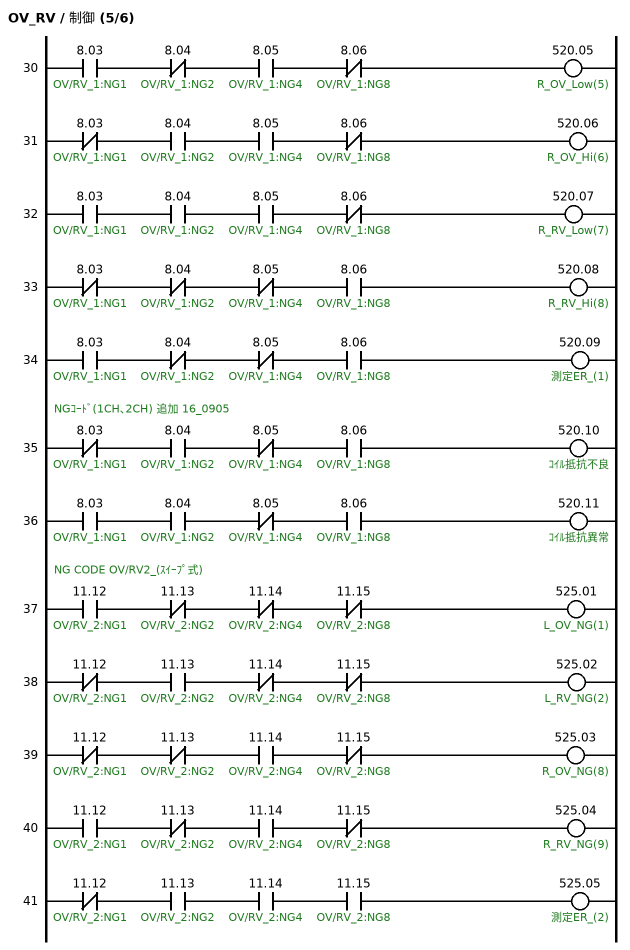
; [picture p120: OV_RV / 制御, rungs 30-41]
; rung 30
LD 8.03  ; OV/RV_1:NG1
ANDNOT 8.04  ; OV/RV_1:NG2
AND 8.05  ; OV/RV_1:NG4
ANDNOT 8.06  ; OV/RV_1:NG8
OUT 520.05  ; R_OV_Low(5)
; rung 31
LDNOT 8.03  ; OV/RV_1:NG1
AND 8.04  ; OV/RV_1:NG2
AND 8.05  ; OV/RV_1:NG4
ANDNOT 8.06  ; OV/RV_1:NG8
OUT 520.06  ; R_OV_Hi(6)
; rung 32
LD 8.03  ; OV/RV_1:NG1
AND 8.04  ; OV/RV_1:NG2
AND 8.05  ; OV/RV_1:NG4
ANDNOT 8.06  ; OV/RV_1:NG8
OUT 520.07  ; R_RV_Low(7)
; rung 33
LDNOT 8.03  ; OV/RV_1:NG1
ANDNOT 8.04  ; OV/RV_1:NG2
ANDNOT 8.05  ; OV/RV_1:NG4
AND 8.06  ; OV/RV_1:NG8
OUT 520.08  ; R_RV_Hi(8)
; rung 34
LD 8.03  ; OV/RV_1:NG1
ANDNOT 8.04  ; OV/RV_1:NG2
ANDNOT 8.05  ; OV/RV_1:NG4
AND 8.06  ; OV/RV_1:NG8
OUT 520.09  ; 測定ER_(1)
; rung 35: NGｺｰﾄﾞ(1CH､2CH) 追加 16_0905
LDNOT 8.03  ; OV/RV_1:NG1
AND 8.04  ; OV/RV_1:NG2
ANDNOT 8.05  ; OV/RV_1:NG4
AND 8.06  ; OV/RV_1:NG8
OUT 520.10  ; ｺｲﾙ抵抗不良
; rung 36
LD 8.03  ; OV/RV_1:NG1
AND 8.04  ; OV/RV_1:NG2
ANDNOT 8.05  ; OV/RV_1:NG4
AND 8.06  ; OV/RV_1:NG8
OUT 520.11  ; ｺｲﾙ抵抗異常
; rung 37: NG CODE OV/RV2_(ｽｲｰﾌﾟ式)
LD 11.12  ; OV/RV_2:NG1
ANDNOT 11.13  ; OV/RV_2:NG2
ANDNOT 11.14  ; OV/RV_2:NG4
ANDNOT 11.15  ; OV/RV_2:NG8
OUT 525.01  ; L_OV_NG(1)
; rung 38
LDNOT 11.12  ; OV/RV_2:NG1
AND 11.13  ; OV/RV_2:NG2
ANDNOT 11.14  ; OV/RV_2:NG4
ANDNOT 11.15  ; OV/RV_2:NG8
OUT 525.02  ; L_RV_NG(2)
; rung 39
LDNOT 11.12  ; OV/RV_2:NG1
ANDNOT 11.13  ; OV/RV_2:NG2
AND 11.14  ; OV/RV_2:NG4
ANDNOT 11.15  ; OV/RV_2:NG8
OUT 525.03  ; R_OV_NG(8)
; rung 40
LD 11.12  ; OV/RV_2:NG1
ANDNOT 11.13  ; OV/RV_2:NG2
AND 11.14  ; OV/RV_2:NG4
ANDNOT 11.15  ; OV/RV_2:NG8
OUT 525.04  ; R_RV_NG(9)
; rung 41
LDNOT 11.12  ; OV/RV_2:NG1
AND 11.13  ; OV/RV_2:NG2
AND 11.14  ; OV/RV_2:NG4
AND 11.15  ; OV/RV_2:NG8
OUT 525.05  ; 測定ER_(2)

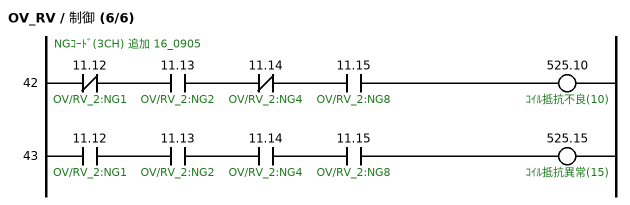
; rung 42: NGｺｰﾄﾞ(3CH) 追加 16_0905
LDNOT 11.12  ; OV/RV_2:NG1
AND 11.13  ; OV/RV_2:NG2
ANDNOT 11.14  ; OV/RV_2:NG4
AND 11.15  ; OV/RV_2:NG8
OUT 525.10  ; ｺｲﾙ抵抗不良(10)
; rung 43
LD 11.12  ; OV/RV_2:NG1
AND 11.13  ; OV/RV_2:NG2
AND 11.14  ; OV/RV_2:NG4
AND 11.15  ; OV/RV_2:NG8
OUT 525.15  ; ｺｲﾙ抵抗異常(15)

### Section 出力

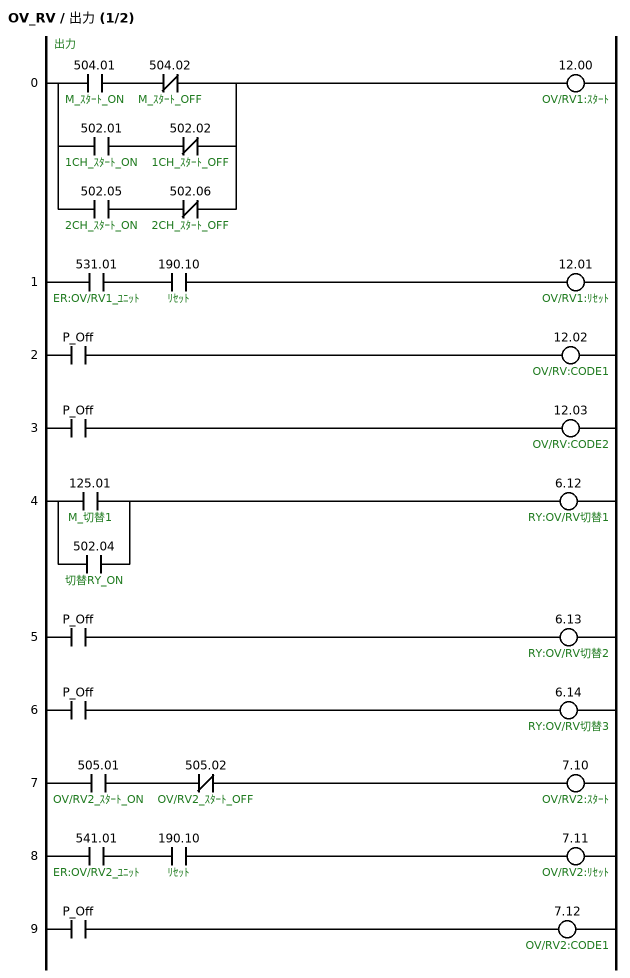
; rung 0: 出力
LD 504.01  ; M_ｽﾀｰﾄ_ON
ANDNOT 504.02  ; M_ｽﾀｰﾄ_OFF
LD 502.01  ; 1CH_ｽﾀｰﾄ_ON
ANDNOT 502.02  ; 1CH_ｽﾀｰﾄ_OFF
ORLD
LD 502.05  ; 2CH_ｽﾀｰﾄ_ON
ANDNOT 502.06  ; 2CH_ｽﾀｰﾄ_OFF
ORLD
OUT 12.00  ; OV/RV1:ｽﾀｰﾄ
; rung 1
LD 531.01  ; ER:OV/RV1_ﾕﾆｯﾄ
AND 190.10  ; ﾘｾｯﾄ
OUT 12.01  ; OV/RV1:ﾘｾｯﾄ
; rung 2
LD P_Off
OUT 12.02  ; OV/RV:CODE1
; rung 3
LD P_Off
OUT 12.03  ; OV/RV:CODE2
; rung 4
LD 125.01  ; M_切替1
OR 502.04  ; 切替RY_ON
OUT 6.12  ; RY:OV/RV切替1
; rung 5
LD P_Off
OUT 6.13  ; RY:OV/RV切替2
; rung 6
LD P_Off
OUT 6.14  ; RY:OV/RV切替3
; rung 7
LD 505.01  ; OV/RV2_ｽﾀｰﾄ_ON
ANDNOT 505.02  ; OV/RV2_ｽﾀｰﾄ_OFF
OUT 7.10  ; OV/RV2:ｽﾀｰﾄ
; rung 8
LD 541.01  ; ER:OV/RV2_ﾕﾆｯﾄ
AND 190.10  ; ﾘｾｯﾄ
OUT 7.11  ; OV/RV2:ﾘｾｯﾄ
; rung 9
LD P_Off
OUT 7.12  ; OV/RV2:CODE1

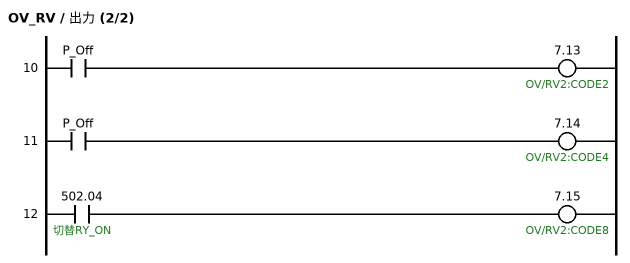
; rung 10
LD P_Off
OUT 7.13  ; OV/RV2:CODE2
; rung 11
LD P_Off
OUT 7.14  ; OV/RV2:CODE4
; rung 12
LD 502.04  ; 切替RY_ON
OUT 7.15  ; OV/RV2:CODE8

### Section ｴﾗｰ

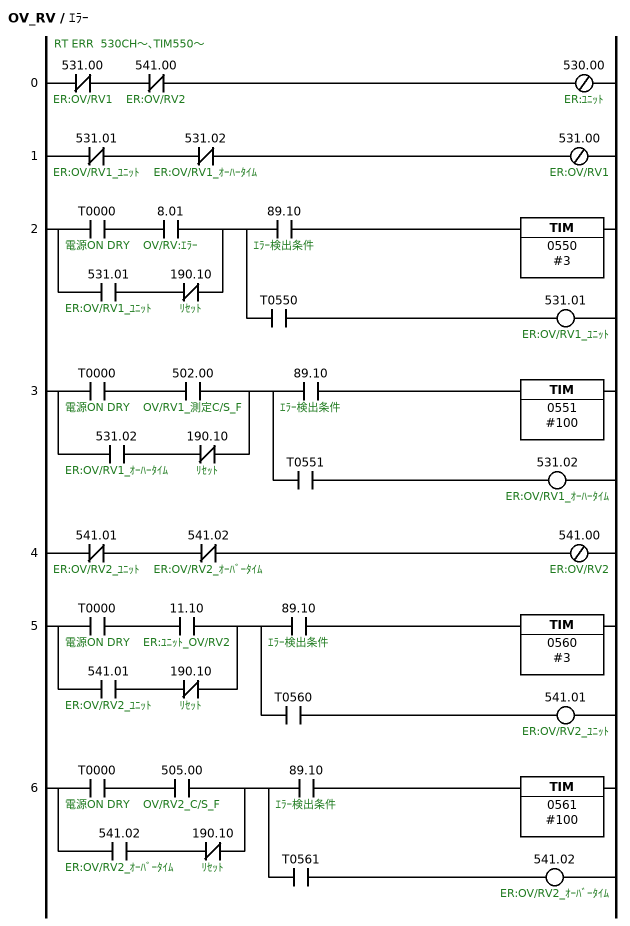
; rung 0: RT ERR  530CH～､TIM550～
LDNOT 531.00  ; ER:OV/RV1
ANDNOT 541.00  ; ER:OV/RV2
OUTNOT 530.00  ; ER:ﾕﾆｯﾄ
; rung 1
LDNOT 531.01  ; ER:OV/RV1_ﾕﾆｯﾄ
ANDNOT 531.02  ; ER:OV/RV1_ｵｰﾊｰﾀｲﾑ
OUTNOT 531.00  ; ER:OV/RV1
; rung 2
LD T0000  ; 電源ON DRY
AND 8.01  ; OV/RV:ｴﾗｰ
LD 531.01  ; ER:OV/RV1_ﾕﾆｯﾄ
ANDNOT 190.10  ; ﾘｾｯﾄ
ORLD
OUT TR0
AND 89.10  ; ｴﾗｰ検出条件
TIM 0550 #3
LD TR0
AND T0550
OUT 531.01  ; ER:OV/RV1_ﾕﾆｯﾄ
; rung 3
LD T0000  ; 電源ON DRY
AND 502.00  ; OV/RV1_測定C/S_F
LD 531.02  ; ER:OV/RV1_ｵｰﾊｰﾀｲﾑ
ANDNOT 190.10  ; ﾘｾｯﾄ
ORLD
OUT TR0
AND 89.10  ; ｴﾗｰ検出条件
TIM 0551 #100
LD TR0
AND T0551
OUT 531.02  ; ER:OV/RV1_ｵｰﾊｰﾀｲﾑ
; rung 4
LDNOT 541.01  ; ER:OV/RV2_ﾕﾆｯﾄ
ANDNOT 541.02  ; ER:OV/RV2_ｵｰﾊﾞｰﾀｲﾑ
OUTNOT 541.00  ; ER:OV/RV2
; rung 5
LD T0000  ; 電源ON DRY
AND 11.10  ; ER:ﾕﾆｯﾄ_OV/RV2
LD 541.01  ; ER:OV/RV2_ﾕﾆｯﾄ
ANDNOT 190.10  ; ﾘｾｯﾄ
ORLD
OUT TR0
AND 89.10  ; ｴﾗｰ検出条件
TIM 0560 #3
LD TR0
AND T0560
OUT 541.01  ; ER:OV/RV2_ﾕﾆｯﾄ
; rung 6
LD T0000  ; 電源ON DRY
AND 505.00  ; OV/RV2_C/S_F
LD 541.02  ; ER:OV/RV2_ｵｰﾊﾞｰﾀｲﾑ
ANDNOT 190.10  ; ﾘｾｯﾄ
ORLD
OUT TR0
AND 89.10  ; ｴﾗｰ検出条件
TIM 0561 #100
LD TR0
AND T0561
OUT 541.02  ; ER:OV/RV2_ｵｰﾊﾞｰﾀｲﾑ

### Section END
; rung 0
END(001)

## Program CP (cyclic task 5)

### Section 制御

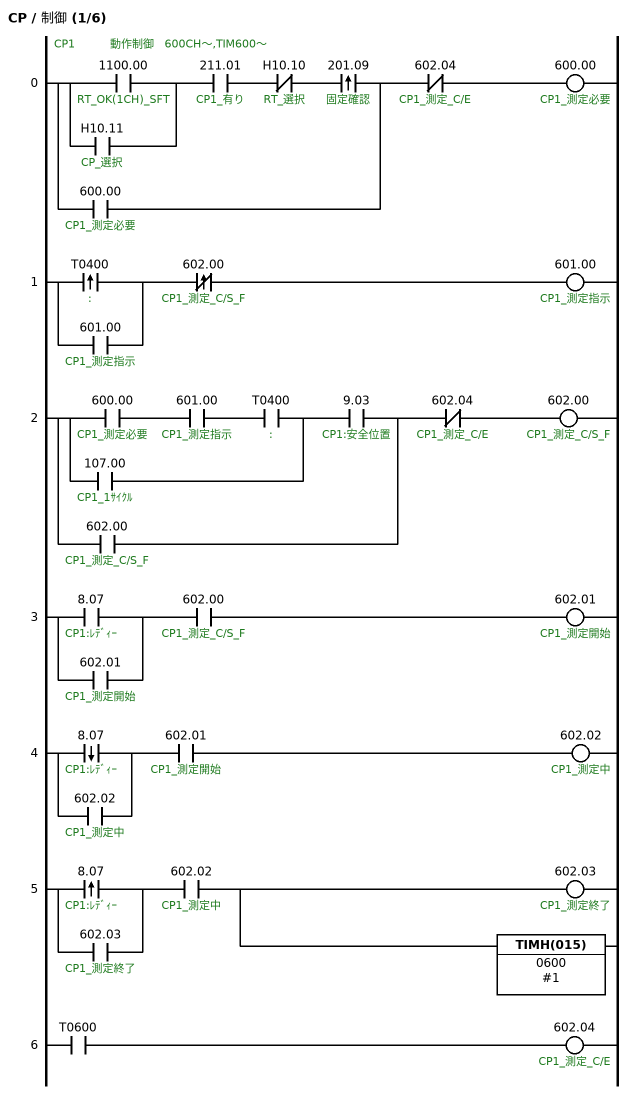
; rung 0: CP1          動作制御   600CH～,TIM600～
LD 1100.00  ; RT_OK(1CH)_SFT
OR H10.11  ; CP_選択
AND 211.01  ; CP1_有り
ANDNOT H10.10  ; RT_選択
@AND 201.09  ; 固定確認
OR 600.00  ; CP1_測定必要
ANDNOT 602.04  ; CP1_測定_C/E
OUT 600.00  ; CP1_測定必要
; rung 1
@LD T0400  ; :
OR 601.00  ; CP1_測定指示
@ANDNOT 602.00  ; CP1_測定_C/S_F
OUT 601.00  ; CP1_測定指示
; rung 2
LD 600.00  ; CP1_測定必要
AND 601.00  ; CP1_測定指示
AND T0400  ; :
OR 107.00  ; CP1_1ｻｲｸﾙ
AND 9.03  ; CP1:安全位置
OR 602.00  ; CP1_測定_C/S_F
ANDNOT 602.04  ; CP1_測定_C/E
OUT 602.00  ; CP1_測定_C/S_F
; rung 3
LD 8.07  ; CP1:ﾚﾃﾞｨｰ
OR 602.01  ; CP1_測定開始
AND 602.00  ; CP1_測定_C/S_F
OUT 602.01  ; CP1_測定開始
; rung 4
%LD 8.07  ; CP1:ﾚﾃﾞｨｰ
OR 602.02  ; CP1_測定中
AND 602.01  ; CP1_測定開始
OUT 602.02  ; CP1_測定中
; rung 5
@LD 8.07  ; CP1:ﾚﾃﾞｨｰ
OR 602.03  ; CP1_測定終了
AND 602.02  ; CP1_測定中
OUT 602.03  ; CP1_測定終了
TIMH(015) 0600 #1
; rung 6
LD T0600
OUT 602.04  ; CP1_測定_C/E

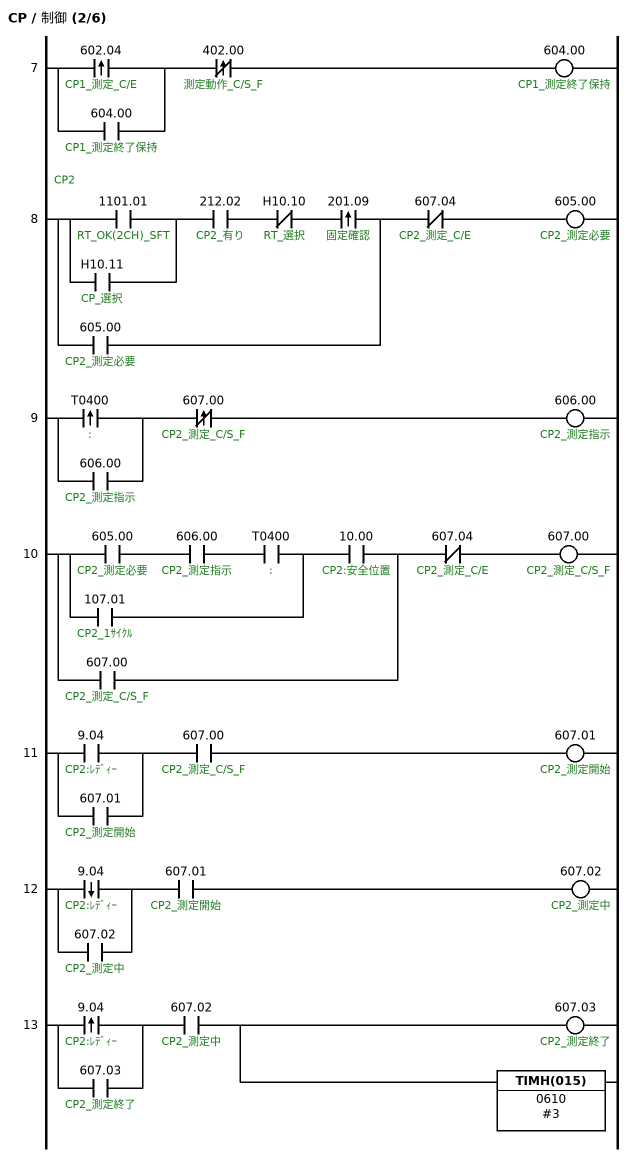
; rung 7
@LD 602.04  ; CP1_測定_C/E
OR 604.00  ; CP1_測定終了保持
@ANDNOT 402.00  ; 測定動作_C/S_F
OUT 604.00  ; CP1_測定終了保持
; rung 8: CP2
LD 1101.01  ; RT_OK(2CH)_SFT
OR H10.11  ; CP_選択
AND 212.02  ; CP2_有り
ANDNOT H10.10  ; RT_選択
@AND 201.09  ; 固定確認
OR 605.00  ; CP2_測定必要
ANDNOT 607.04  ; CP2_測定_C/E
OUT 605.00  ; CP2_測定必要
; rung 9
@LD T0400  ; :
OR 606.00  ; CP2_測定指示
@ANDNOT 607.00  ; CP2_測定_C/S_F
OUT 606.00  ; CP2_測定指示
; rung 10
LD 605.00  ; CP2_測定必要
AND 606.00  ; CP2_測定指示
AND T0400  ; :
OR 107.01  ; CP2_1ｻｲｸﾙ
AND 10.00  ; CP2:安全位置
OR 607.00  ; CP2_測定_C/S_F
ANDNOT 607.04  ; CP2_測定_C/E
OUT 607.00  ; CP2_測定_C/S_F
; rung 11
LD 9.04  ; CP2:ﾚﾃﾞｨｰ
OR 607.01  ; CP2_測定開始
AND 607.00  ; CP2_測定_C/S_F
OUT 607.01  ; CP2_測定開始
; rung 12
%LD 9.04  ; CP2:ﾚﾃﾞｨｰ
OR 607.02  ; CP2_測定中
AND 607.01  ; CP2_測定開始
OUT 607.02  ; CP2_測定中
; rung 13
@LD 9.04  ; CP2:ﾚﾃﾞｨｰ
OR 607.03  ; CP2_測定終了
AND 607.02  ; CP2_測定中
OUT 607.03  ; CP2_測定終了
TIMH(015) 0610 #3

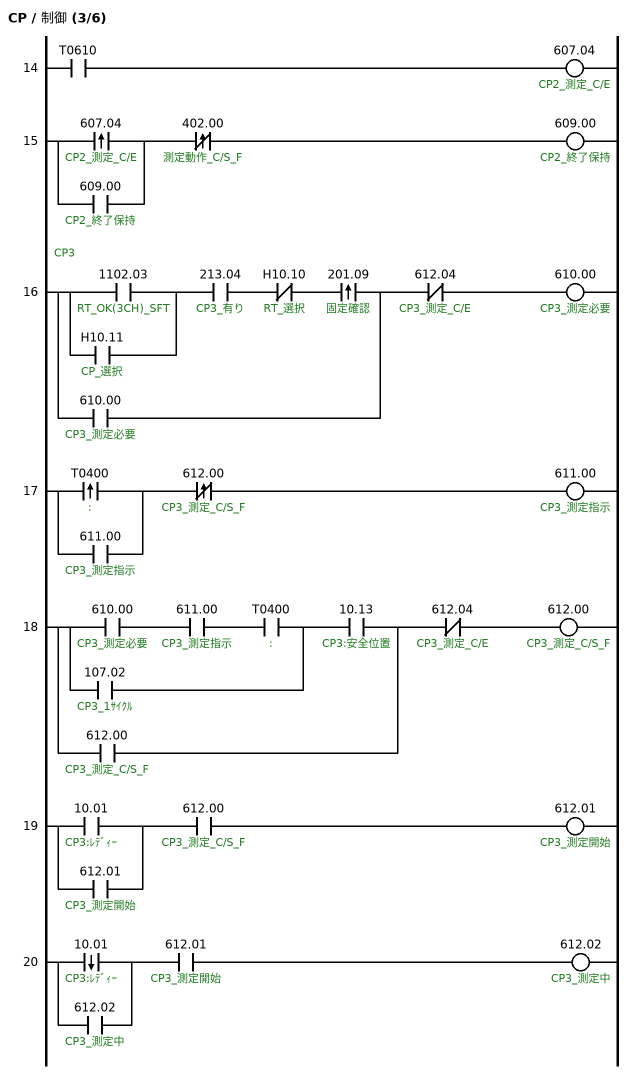
; rung 14
LD T0610
OUT 607.04  ; CP2_測定_C/E
; rung 15
@LD 607.04  ; CP2_測定_C/E
OR 609.00  ; CP2_終了保持
@ANDNOT 402.00  ; 測定動作_C/S_F
OUT 609.00  ; CP2_終了保持
; rung 16: CP3
LD 1102.03  ; RT_OK(3CH)_SFT
OR H10.11  ; CP_選択
AND 213.04  ; CP3_有り
ANDNOT H10.10  ; RT_選択
@AND 201.09  ; 固定確認
OR 610.00  ; CP3_測定必要
ANDNOT 612.04  ; CP3_測定_C/E
OUT 610.00  ; CP3_測定必要
; rung 17
@LD T0400  ; :
OR 611.00  ; CP3_測定指示
@ANDNOT 612.00  ; CP3_測定_C/S_F
OUT 611.00  ; CP3_測定指示
; rung 18
LD 610.00  ; CP3_測定必要
AND 611.00  ; CP3_測定指示
AND T0400  ; :
OR 107.02  ; CP3_1ｻｲｸﾙ
AND 10.13  ; CP3:安全位置
OR 612.00  ; CP3_測定_C/S_F
ANDNOT 612.04  ; CP3_測定_C/E
OUT 612.00  ; CP3_測定_C/S_F
; rung 19
LD 10.01  ; CP3:ﾚﾃﾞｨｰ
OR 612.01  ; CP3_測定開始
AND 612.00  ; CP3_測定_C/S_F
OUT 612.01  ; CP3_測定開始
; rung 20
%LD 10.01  ; CP3:ﾚﾃﾞｨｰ
OR 612.02  ; CP3_測定中
AND 612.01  ; CP3_測定開始
OUT 612.02  ; CP3_測定中

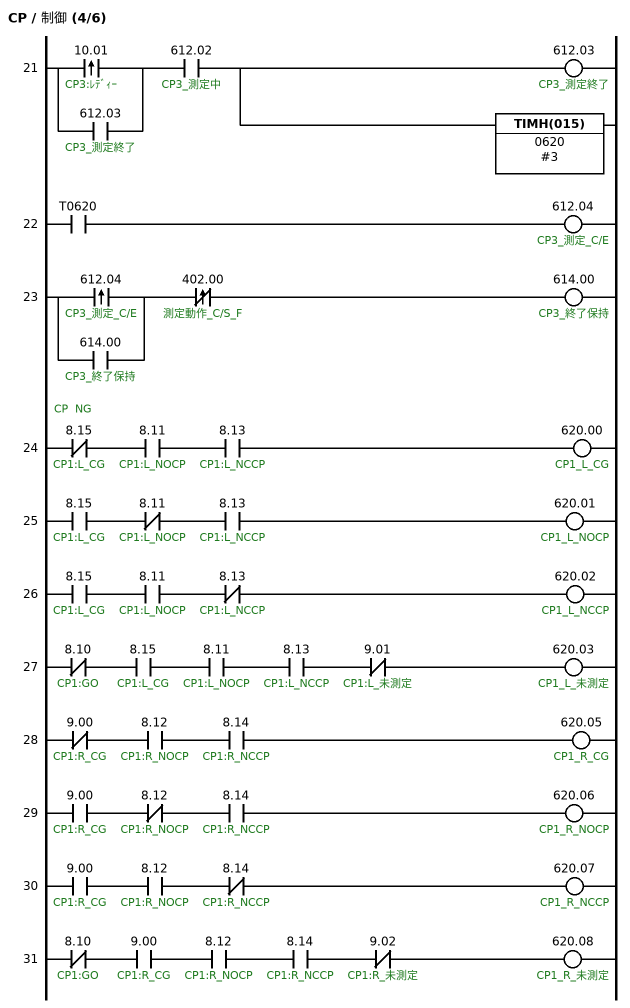
; rung 21
@LD 10.01  ; CP3:ﾚﾃﾞｨｰ
OR 612.03  ; CP3_測定終了
AND 612.02  ; CP3_測定中
OUT 612.03  ; CP3_測定終了
TIMH(015) 0620 #3
; rung 22
LD T0620
OUT 612.04  ; CP3_測定_C/E
; rung 23
@LD 612.04  ; CP3_測定_C/E
OR 614.00  ; CP3_終了保持
@ANDNOT 402.00  ; 測定動作_C/S_F
OUT 614.00  ; CP3_終了保持
; rung 24: CP  NG
LDNOT 8.15  ; CP1:L_CG
AND 8.11  ; CP1:L_NOCP
AND 8.13  ; CP1:L_NCCP
OUT 620.00  ; CP1_L_CG
; rung 25
LD 8.15  ; CP1:L_CG
ANDNOT 8.11  ; CP1:L_NOCP
AND 8.13  ; CP1:L_NCCP
OUT 620.01  ; CP1_L_NOCP
; rung 26
LD 8.15  ; CP1:L_CG
AND 8.11  ; CP1:L_NOCP
ANDNOT 8.13  ; CP1:L_NCCP
OUT 620.02  ; CP1_L_NCCP
; rung 27
LDNOT 8.10  ; CP1:GO
AND 8.15  ; CP1:L_CG
AND 8.11  ; CP1:L_NOCP
AND 8.13  ; CP1:L_NCCP
ANDNOT 9.01  ; CP1:L_未測定
OUT 620.03  ; CP1_L_未測定
; rung 28
LDNOT 9.00  ; CP1:R_CG
AND 8.12  ; CP1:R_NOCP
AND 8.14  ; CP1:R_NCCP
OUT 620.05  ; CP1_R_CG
; rung 29
LD 9.00  ; CP1:R_CG
ANDNOT 8.12  ; CP1:R_NOCP
AND 8.14  ; CP1:R_NCCP
OUT 620.06  ; CP1_R_NOCP
; rung 30
LD 9.00  ; CP1:R_CG
AND 8.12  ; CP1:R_NOCP
ANDNOT 8.14  ; CP1:R_NCCP
OUT 620.07  ; CP1_R_NCCP
; rung 31
LDNOT 8.10  ; CP1:GO
AND 9.00  ; CP1:R_CG
AND 8.12  ; CP1:R_NOCP
AND 8.14  ; CP1:R_NCCP
ANDNOT 9.02  ; CP1:R_未測定
OUT 620.08  ; CP1_R_未測定

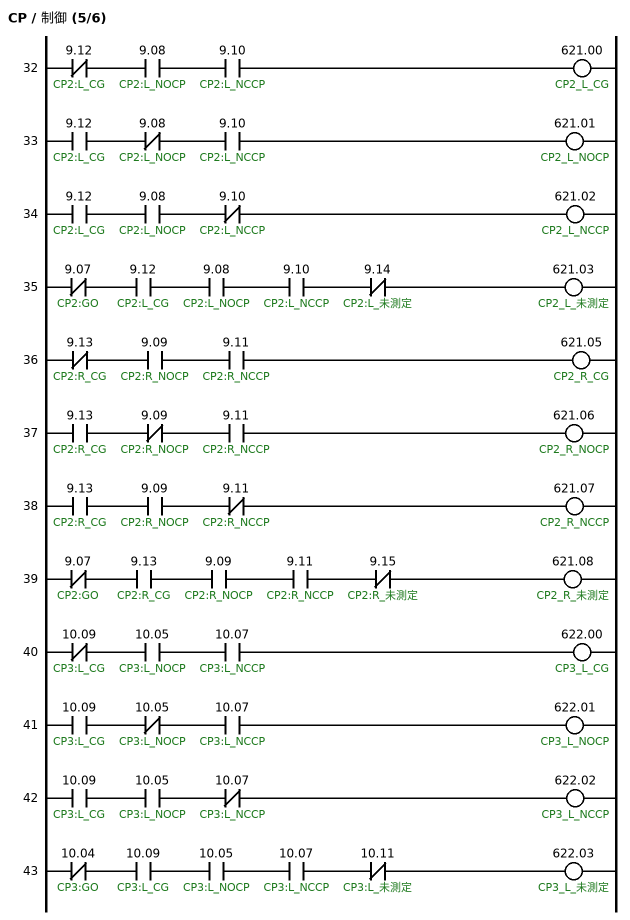
; rung 32
LDNOT 9.12  ; CP2:L_CG
AND 9.08  ; CP2:L_NOCP
AND 9.10  ; CP2:L_NCCP
OUT 621.00  ; CP2_L_CG
; rung 33
LD 9.12  ; CP2:L_CG
ANDNOT 9.08  ; CP2:L_NOCP
AND 9.10  ; CP2:L_NCCP
OUT 621.01  ; CP2_L_NOCP
; rung 34
LD 9.12  ; CP2:L_CG
AND 9.08  ; CP2:L_NOCP
ANDNOT 9.10  ; CP2:L_NCCP
OUT 621.02  ; CP2_L_NCCP
; rung 35
LDNOT 9.07  ; CP2:GO
AND 9.12  ; CP2:L_CG
AND 9.08  ; CP2:L_NOCP
AND 9.10  ; CP2:L_NCCP
ANDNOT 9.14  ; CP2:L_未測定
OUT 621.03  ; CP2_L_未測定
; rung 36
LDNOT 9.13  ; CP2:R_CG
AND 9.09  ; CP2:R_NOCP
AND 9.11  ; CP2:R_NCCP
OUT 621.05  ; CP2_R_CG
; rung 37
LD 9.13  ; CP2:R_CG
ANDNOT 9.09  ; CP2:R_NOCP
AND 9.11  ; CP2:R_NCCP
OUT 621.06  ; CP2_R_NOCP
; rung 38
LD 9.13  ; CP2:R_CG
AND 9.09  ; CP2:R_NOCP
ANDNOT 9.11  ; CP2:R_NCCP
OUT 621.07  ; CP2_R_NCCP
; rung 39
LDNOT 9.07  ; CP2:GO
AND 9.13  ; CP2:R_CG
AND 9.09  ; CP2:R_NOCP
AND 9.11  ; CP2:R_NCCP
ANDNOT 9.15  ; CP2:R_未測定
OUT 621.08  ; CP2_R_未測定
; rung 40
LDNOT 10.09  ; CP3:L_CG
AND 10.05  ; CP3:L_NOCP
AND 10.07  ; CP3:L_NCCP
OUT 622.00  ; CP3_L_CG
; rung 41
LD 10.09  ; CP3:L_CG
ANDNOT 10.05  ; CP3:L_NOCP
AND 10.07  ; CP3:L_NCCP
OUT 622.01  ; CP3_L_NOCP
; rung 42
LD 10.09  ; CP3:L_CG
AND 10.05  ; CP3:L_NOCP
ANDNOT 10.07  ; CP3:L_NCCP
OUT 622.02  ; CP3_L_NCCP
; rung 43
LDNOT 10.04  ; CP3:GO
AND 10.09  ; CP3:L_CG
AND 10.05  ; CP3:L_NOCP
AND 10.07  ; CP3:L_NCCP
ANDNOT 10.11  ; CP3:L_未測定
OUT 622.03  ; CP3_L_未測定

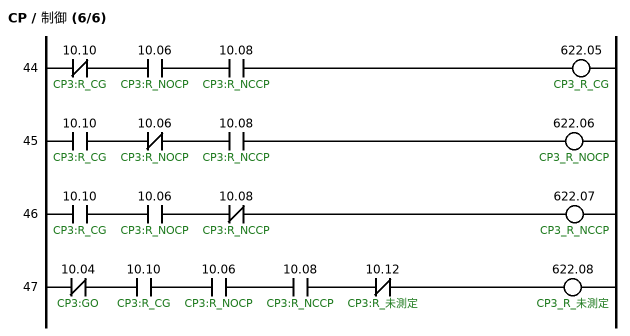
; rung 44
LDNOT 10.10  ; CP3:R_CG
AND 10.06  ; CP3:R_NOCP
AND 10.08  ; CP3:R_NCCP
OUT 622.05  ; CP3_R_CG
; rung 45
LD 10.10  ; CP3:R_CG
ANDNOT 10.06  ; CP3:R_NOCP
AND 10.08  ; CP3:R_NCCP
OUT 622.06  ; CP3_R_NOCP
; rung 46
LD 10.10  ; CP3:R_CG
AND 10.06  ; CP3:R_NOCP
ANDNOT 10.08  ; CP3:R_NCCP
OUT 622.07  ; CP3_R_NCCP
; rung 47
LDNOT 10.04  ; CP3:GO
AND 10.10  ; CP3:R_CG
AND 10.06  ; CP3:R_NOCP
AND 10.08  ; CP3:R_NCCP
ANDNOT 10.12  ; CP3:R_未測定
OUT 622.08  ; CP3_R_未測定

### Section 出力

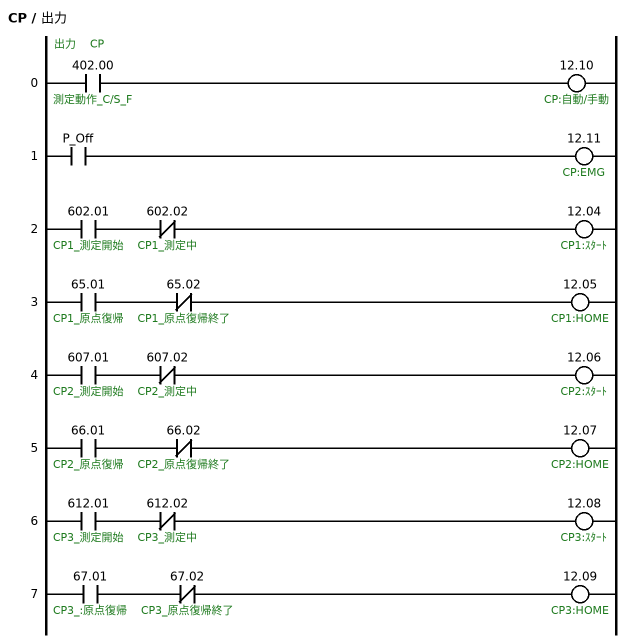
; rung 0: 出力    CP
LD 402.00  ; 測定動作_C/S_F
OUT 12.10  ; CP:自動/手動
; rung 1
LD P_Off
OUT 12.11  ; CP:EMG
; rung 2
LD 602.01  ; CP1_測定開始
ANDNOT 602.02  ; CP1_測定中
OUT 12.04  ; CP1:ｽﾀｰﾄ
; rung 3
LD 65.01  ; CP1_原点復帰
ANDNOT 65.02  ; CP1_原点復帰終了
OUT 12.05  ; CP1:HOME
; rung 4
LD 607.01  ; CP2_測定開始
ANDNOT 607.02  ; CP2_測定中
OUT 12.06  ; CP2:ｽﾀｰﾄ
; rung 5
LD 66.01  ; CP2_原点復帰
ANDNOT 66.02  ; CP2_原点復帰終了
OUT 12.07  ; CP2:HOME
; rung 6
LD 612.01  ; CP3_測定開始
ANDNOT 612.02  ; CP3_測定中
OUT 12.08  ; CP3:ｽﾀｰﾄ
; rung 7
LD 67.01  ; CP3_:原点復帰
ANDNOT 67.02  ; CP3_原点復帰終了
OUT 12.09  ; CP3:HOME

### Section ｴﾗｰ

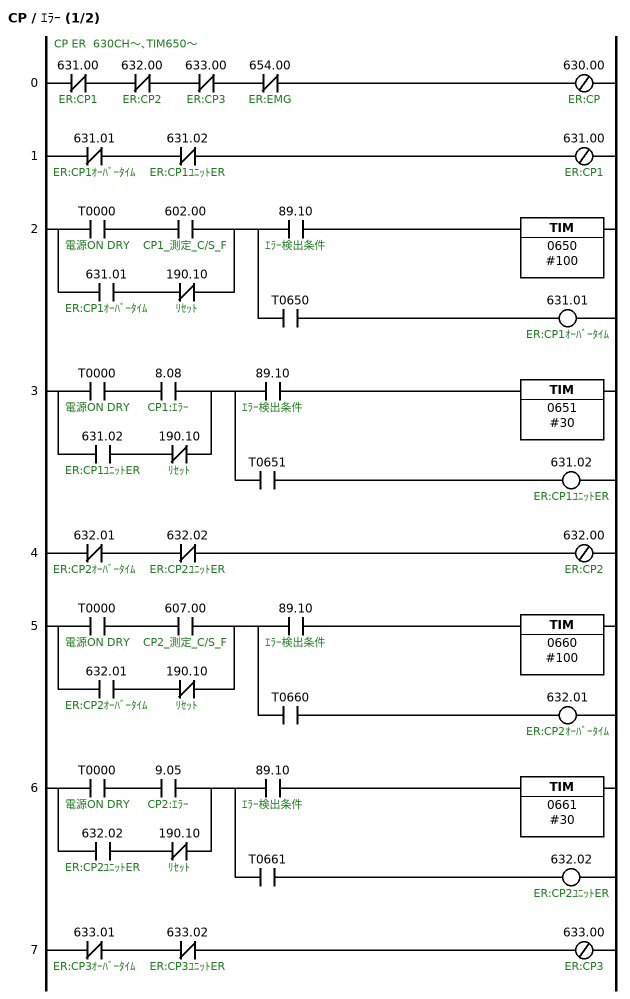
; rung 0: CP ER  630CH～､TIM650～
LDNOT 631.00  ; ER:CP1
ANDNOT 632.00  ; ER:CP2
ANDNOT 633.00  ; ER:CP3
ANDNOT 654.00  ; ER:EMG
OUTNOT 630.00  ; ER:CP
; rung 1
LDNOT 631.01  ; ER:CP1ｵｰﾊﾞｰﾀｲﾑ
ANDNOT 631.02  ; ER:CP1ﾕﾆｯﾄER
OUTNOT 631.00  ; ER:CP1
; rung 2
LD T0000  ; 電源ON DRY
AND 602.00  ; CP1_測定_C/S_F
LD 631.01  ; ER:CP1ｵｰﾊﾞｰﾀｲﾑ
ANDNOT 190.10  ; ﾘｾｯﾄ
ORLD
OUT TR0
AND 89.10  ; ｴﾗｰ検出条件
TIM 0650 #100
LD TR0
AND T0650
OUT 631.01  ; ER:CP1ｵｰﾊﾞｰﾀｲﾑ
; rung 3
LD T0000  ; 電源ON DRY
AND 8.08  ; CP1:ｴﾗｰ
LD 631.02  ; ER:CP1ﾕﾆｯﾄER
ANDNOT 190.10  ; ﾘｾｯﾄ
ORLD
OUT TR0
AND 89.10  ; ｴﾗｰ検出条件
TIM 0651 #30
LD TR0
AND T0651
OUT 631.02  ; ER:CP1ﾕﾆｯﾄER
; rung 4
LDNOT 632.01  ; ER:CP2ｵｰﾊﾞｰﾀｲﾑ
ANDNOT 632.02  ; ER:CP2ﾕﾆｯﾄER
OUTNOT 632.00  ; ER:CP2
; rung 5
LD T0000  ; 電源ON DRY
AND 607.00  ; CP2_測定_C/S_F
LD 632.01  ; ER:CP2ｵｰﾊﾞｰﾀｲﾑ
ANDNOT 190.10  ; ﾘｾｯﾄ
ORLD
OUT TR0
AND 89.10  ; ｴﾗｰ検出条件
TIM 0660 #100
LD TR0
AND T0660
OUT 632.01  ; ER:CP2ｵｰﾊﾞｰﾀｲﾑ
; rung 6
LD T0000  ; 電源ON DRY
AND 9.05  ; CP2:ｴﾗｰ
LD 632.02  ; ER:CP2ﾕﾆｯﾄER
ANDNOT 190.10  ; ﾘｾｯﾄ
ORLD
OUT TR0
AND 89.10  ; ｴﾗｰ検出条件
TIM 0661 #30
LD TR0
AND T0661
OUT 632.02  ; ER:CP2ﾕﾆｯﾄER
; rung 7
LDNOT 633.01  ; ER:CP3ｵｰﾊﾞｰﾀｲﾑ
ANDNOT 633.02  ; ER:CP3ﾕﾆｯﾄER
OUTNOT 633.00  ; ER:CP3

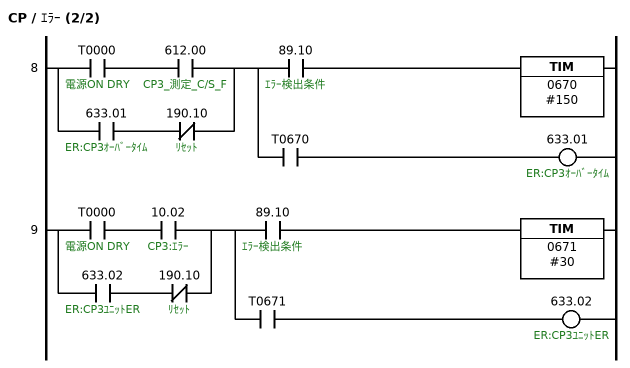
; rung 8
LD T0000  ; 電源ON DRY
AND 612.00  ; CP3_測定_C/S_F
LD 633.01  ; ER:CP3ｵｰﾊﾞｰﾀｲﾑ
ANDNOT 190.10  ; ﾘｾｯﾄ
ORLD
OUT TR0
AND 89.10  ; ｴﾗｰ検出条件
TIM 0670 #150
LD TR0
AND T0670
OUT 633.01  ; ER:CP3ｵｰﾊﾞｰﾀｲﾑ
; rung 9
LD T0000  ; 電源ON DRY
AND 10.02  ; CP3:ｴﾗｰ
LD 633.02  ; ER:CP3ﾕﾆｯﾄER
ANDNOT 190.10  ; ﾘｾｯﾄ
ORLD
OUT TR0
AND 89.10  ; ｴﾗｰ検出条件
TIM 0671 #30
LD TR0
AND T0671
OUT 633.02  ; ER:CP3ﾕﾆｯﾄER

### Section END
; rung 0
END(001)

## Program ﾃｰﾀ処理 (cyclic task 6)

### Section 判定保持

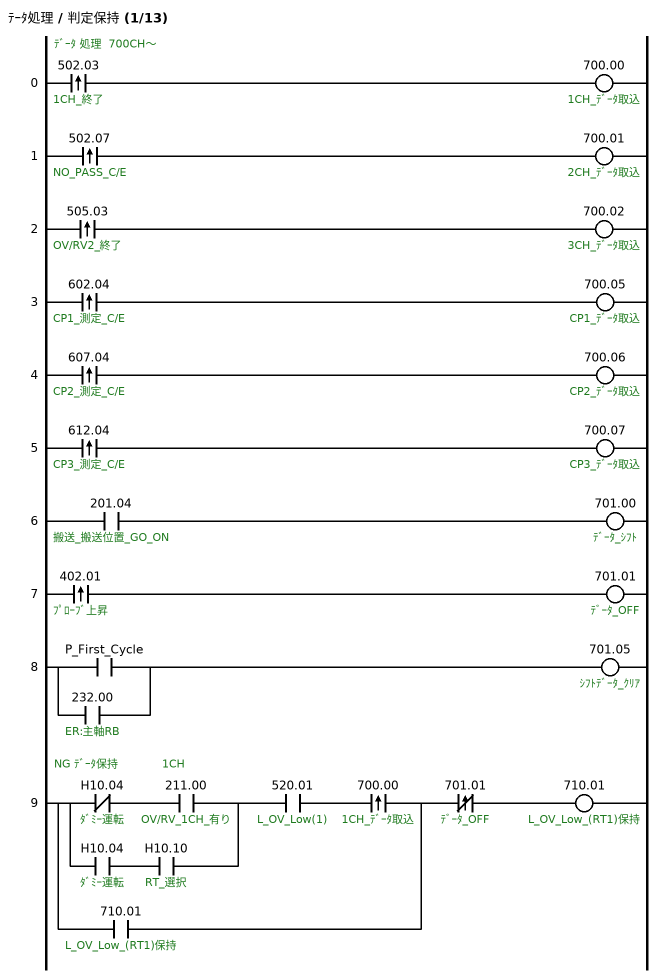
; rung 0: ﾃﾞｰﾀ 処理  700CH～
@LD 502.03  ; 1CH_終了
OUT 700.00  ; 1CH_ﾃﾞｰﾀ取込
; rung 1
@LD 502.07  ; NO_PASS_C/E
OUT 700.01  ; 2CH_ﾃﾞｰﾀ取込
; rung 2
@LD 505.03  ; OV/RV2_終了
OUT 700.02  ; 3CH_ﾃﾞｰﾀ取込
; rung 3
@LD 602.04  ; CP1_測定_C/E
OUT 700.05  ; CP1_ﾃﾞｰﾀ取込
; rung 4
@LD 607.04  ; CP2_測定_C/E
OUT 700.06  ; CP2_ﾃﾞｰﾀ取込
; rung 5
@LD 612.04  ; CP3_測定_C/E
OUT 700.07  ; CP3_ﾃﾞｰﾀ取込
; rung 6
LD 201.04  ; 搬送_搬送位置_GO_ON
OUT 701.00  ; ﾃﾞｰﾀ_ｼﾌﾄ
; rung 7
@LD 402.01  ; ﾌﾟﾛｰﾌﾞ上昇
OUT 701.01  ; ﾃﾞｰﾀ_OFF
; rung 8
LD P_First_Cycle
OR 232.00  ; ER:主軸RB
OUT 701.05  ; ｼﾌﾄﾃﾞｰﾀ_ｸﾘｱ
; rung 9: NG ﾃﾞｰﾀ保持　　　　1CH
LDNOT H10.04  ; ﾀﾞﾐｰ運転
AND 211.00  ; OV/RV_1CH_有り
LD H10.04  ; ﾀﾞﾐｰ運転
AND H10.10  ; RT_選択
ORLD
AND 520.01  ; L_OV_Low(1)
@AND 700.00  ; 1CH_ﾃﾞｰﾀ取込
OR 710.01  ; L_OV_Low_(RT1)保持
@ANDNOT 701.01  ; ﾃﾞｰﾀ_OFF
OUT 710.01  ; L_OV_Low_(RT1)保持

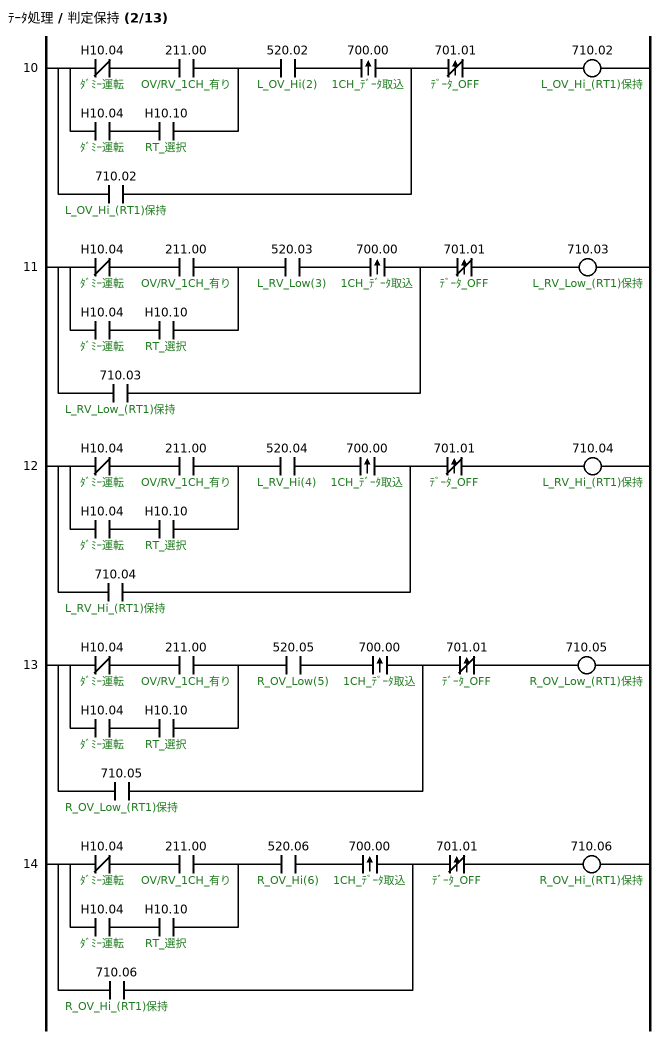
; rung 10
LDNOT H10.04  ; ﾀﾞﾐｰ運転
AND 211.00  ; OV/RV_1CH_有り
LD H10.04  ; ﾀﾞﾐｰ運転
AND H10.10  ; RT_選択
ORLD
AND 520.02  ; L_OV_Hi(2)
@AND 700.00  ; 1CH_ﾃﾞｰﾀ取込
OR 710.02  ; L_OV_Hi_(RT1)保持
@ANDNOT 701.01  ; ﾃﾞｰﾀ_OFF
OUT 710.02  ; L_OV_Hi_(RT1)保持
; rung 11
LDNOT H10.04  ; ﾀﾞﾐｰ運転
AND 211.00  ; OV/RV_1CH_有り
LD H10.04  ; ﾀﾞﾐｰ運転
AND H10.10  ; RT_選択
ORLD
AND 520.03  ; L_RV_Low(3)
@AND 700.00  ; 1CH_ﾃﾞｰﾀ取込
OR 710.03  ; L_RV_Low_(RT1)保持
@ANDNOT 701.01  ; ﾃﾞｰﾀ_OFF
OUT 710.03  ; L_RV_Low_(RT1)保持
; rung 12
LDNOT H10.04  ; ﾀﾞﾐｰ運転
AND 211.00  ; OV/RV_1CH_有り
LD H10.04  ; ﾀﾞﾐｰ運転
AND H10.10  ; RT_選択
ORLD
AND 520.04  ; L_RV_Hi(4)
@AND 700.00  ; 1CH_ﾃﾞｰﾀ取込
OR 710.04  ; L_RV_Hi_(RT1)保持
@ANDNOT 701.01  ; ﾃﾞｰﾀ_OFF
OUT 710.04  ; L_RV_Hi_(RT1)保持
; rung 13
LDNOT H10.04  ; ﾀﾞﾐｰ運転
AND 211.00  ; OV/RV_1CH_有り
LD H10.04  ; ﾀﾞﾐｰ運転
AND H10.10  ; RT_選択
ORLD
AND 520.05  ; R_OV_Low(5)
@AND 700.00  ; 1CH_ﾃﾞｰﾀ取込
OR 710.05  ; R_OV_Low_(RT1)保持
@ANDNOT 701.01  ; ﾃﾞｰﾀ_OFF
OUT 710.05  ; R_OV_Low_(RT1)保持
; rung 14
LDNOT H10.04  ; ﾀﾞﾐｰ運転
AND 211.00  ; OV/RV_1CH_有り
LD H10.04  ; ﾀﾞﾐｰ運転
AND H10.10  ; RT_選択
ORLD
AND 520.06  ; R_OV_Hi(6)
@AND 700.00  ; 1CH_ﾃﾞｰﾀ取込
OR 710.06  ; R_OV_Hi_(RT1)保持
@ANDNOT 701.01  ; ﾃﾞｰﾀ_OFF
OUT 710.06  ; R_OV_Hi_(RT1)保持

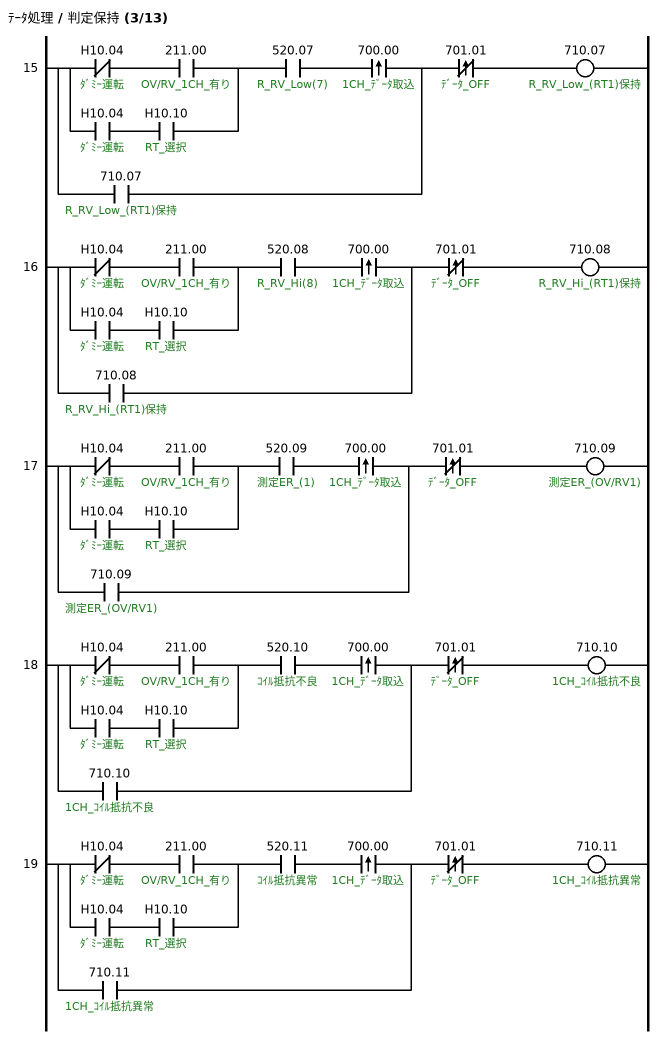
; rung 15
LDNOT H10.04  ; ﾀﾞﾐｰ運転
AND 211.00  ; OV/RV_1CH_有り
LD H10.04  ; ﾀﾞﾐｰ運転
AND H10.10  ; RT_選択
ORLD
AND 520.07  ; R_RV_Low(7)
@AND 700.00  ; 1CH_ﾃﾞｰﾀ取込
OR 710.07  ; R_RV_Low_(RT1)保持
@ANDNOT 701.01  ; ﾃﾞｰﾀ_OFF
OUT 710.07  ; R_RV_Low_(RT1)保持
; rung 16
LDNOT H10.04  ; ﾀﾞﾐｰ運転
AND 211.00  ; OV/RV_1CH_有り
LD H10.04  ; ﾀﾞﾐｰ運転
AND H10.10  ; RT_選択
ORLD
AND 520.08  ; R_RV_Hi(8)
@AND 700.00  ; 1CH_ﾃﾞｰﾀ取込
OR 710.08  ; R_RV_Hi_(RT1)保持
@ANDNOT 701.01  ; ﾃﾞｰﾀ_OFF
OUT 710.08  ; R_RV_Hi_(RT1)保持
; rung 17
LDNOT H10.04  ; ﾀﾞﾐｰ運転
AND 211.00  ; OV/RV_1CH_有り
LD H10.04  ; ﾀﾞﾐｰ運転
AND H10.10  ; RT_選択
ORLD
AND 520.09  ; 測定ER_(1)
@AND 700.00  ; 1CH_ﾃﾞｰﾀ取込
OR 710.09  ; 測定ER_(OV/RV1)
@ANDNOT 701.01  ; ﾃﾞｰﾀ_OFF
OUT 710.09  ; 測定ER_(OV/RV1)
; rung 18
LDNOT H10.04  ; ﾀﾞﾐｰ運転
AND 211.00  ; OV/RV_1CH_有り
LD H10.04  ; ﾀﾞﾐｰ運転
AND H10.10  ; RT_選択
ORLD
AND 520.10  ; ｺｲﾙ抵抗不良
@AND 700.00  ; 1CH_ﾃﾞｰﾀ取込
OR 710.10  ; 1CH_ｺｲﾙ抵抗不良
@ANDNOT 701.01  ; ﾃﾞｰﾀ_OFF
OUT 710.10  ; 1CH_ｺｲﾙ抵抗不良
; rung 19
LDNOT H10.04  ; ﾀﾞﾐｰ運転
AND 211.00  ; OV/RV_1CH_有り
LD H10.04  ; ﾀﾞﾐｰ運転
AND H10.10  ; RT_選択
ORLD
AND 520.11  ; ｺｲﾙ抵抗異常
@AND 700.00  ; 1CH_ﾃﾞｰﾀ取込
OR 710.11  ; 1CH_ｺｲﾙ抵抗異常
@ANDNOT 701.01  ; ﾃﾞｰﾀ_OFF
OUT 710.11  ; 1CH_ｺｲﾙ抵抗異常

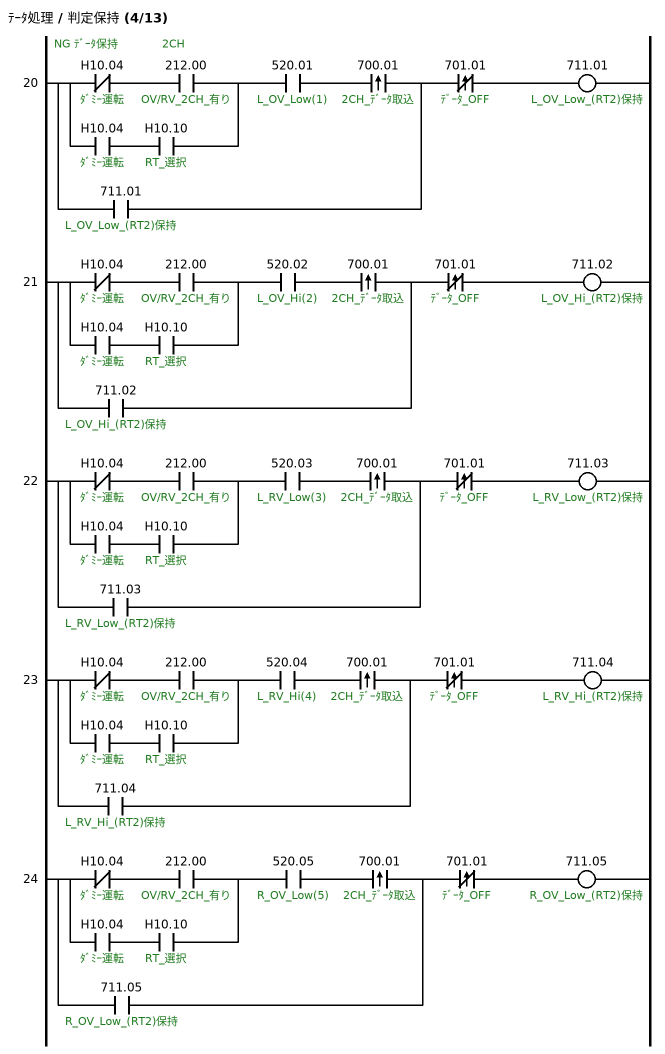
; rung 20: NG ﾃﾞｰﾀ保持　　　　2CH
LDNOT H10.04  ; ﾀﾞﾐｰ運転
AND 212.00  ; OV/RV_2CH_有り
LD H10.04  ; ﾀﾞﾐｰ運転
AND H10.10  ; RT_選択
ORLD
AND 520.01  ; L_OV_Low(1)
@AND 700.01  ; 2CH_ﾃﾞｰﾀ取込
OR 711.01  ; L_OV_Low_(RT2)保持
@ANDNOT 701.01  ; ﾃﾞｰﾀ_OFF
OUT 711.01  ; L_OV_Low_(RT2)保持
; rung 21
LDNOT H10.04  ; ﾀﾞﾐｰ運転
AND 212.00  ; OV/RV_2CH_有り
LD H10.04  ; ﾀﾞﾐｰ運転
AND H10.10  ; RT_選択
ORLD
AND 520.02  ; L_OV_Hi(2)
@AND 700.01  ; 2CH_ﾃﾞｰﾀ取込
OR 711.02  ; L_OV_Hi_(RT2)保持
@ANDNOT 701.01  ; ﾃﾞｰﾀ_OFF
OUT 711.02  ; L_OV_Hi_(RT2)保持
; rung 22
LDNOT H10.04  ; ﾀﾞﾐｰ運転
AND 212.00  ; OV/RV_2CH_有り
LD H10.04  ; ﾀﾞﾐｰ運転
AND H10.10  ; RT_選択
ORLD
AND 520.03  ; L_RV_Low(3)
@AND 700.01  ; 2CH_ﾃﾞｰﾀ取込
OR 711.03  ; L_RV_Low_(RT2)保持
@ANDNOT 701.01  ; ﾃﾞｰﾀ_OFF
OUT 711.03  ; L_RV_Low_(RT2)保持
; rung 23
LDNOT H10.04  ; ﾀﾞﾐｰ運転
AND 212.00  ; OV/RV_2CH_有り
LD H10.04  ; ﾀﾞﾐｰ運転
AND H10.10  ; RT_選択
ORLD
AND 520.04  ; L_RV_Hi(4)
@AND 700.01  ; 2CH_ﾃﾞｰﾀ取込
OR 711.04  ; L_RV_Hi_(RT2)保持
@ANDNOT 701.01  ; ﾃﾞｰﾀ_OFF
OUT 711.04  ; L_RV_Hi_(RT2)保持
; rung 24
LDNOT H10.04  ; ﾀﾞﾐｰ運転
AND 212.00  ; OV/RV_2CH_有り
LD H10.04  ; ﾀﾞﾐｰ運転
AND H10.10  ; RT_選択
ORLD
AND 520.05  ; R_OV_Low(5)
@AND 700.01  ; 2CH_ﾃﾞｰﾀ取込
OR 711.05  ; R_OV_Low_(RT2)保持
@ANDNOT 701.01  ; ﾃﾞｰﾀ_OFF
OUT 711.05  ; R_OV_Low_(RT2)保持

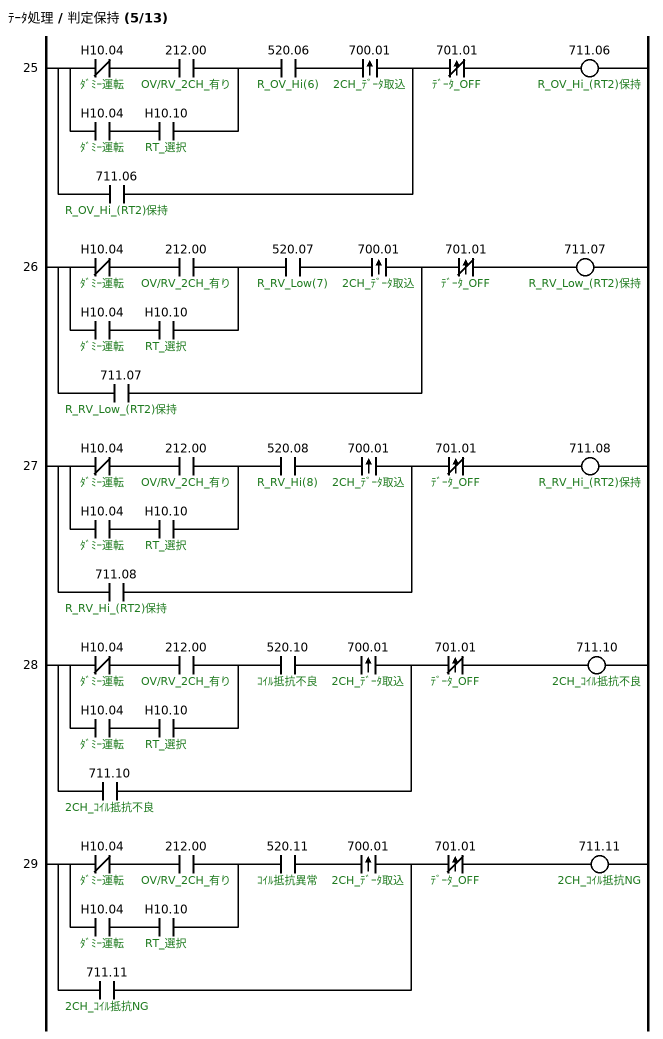
; rung 25
LDNOT H10.04  ; ﾀﾞﾐｰ運転
AND 212.00  ; OV/RV_2CH_有り
LD H10.04  ; ﾀﾞﾐｰ運転
AND H10.10  ; RT_選択
ORLD
AND 520.06  ; R_OV_Hi(6)
@AND 700.01  ; 2CH_ﾃﾞｰﾀ取込
OR 711.06  ; R_OV_Hi_(RT2)保持
@ANDNOT 701.01  ; ﾃﾞｰﾀ_OFF
OUT 711.06  ; R_OV_Hi_(RT2)保持
; rung 26
LDNOT H10.04  ; ﾀﾞﾐｰ運転
AND 212.00  ; OV/RV_2CH_有り
LD H10.04  ; ﾀﾞﾐｰ運転
AND H10.10  ; RT_選択
ORLD
AND 520.07  ; R_RV_Low(7)
@AND 700.01  ; 2CH_ﾃﾞｰﾀ取込
OR 711.07  ; R_RV_Low_(RT2)保持
@ANDNOT 701.01  ; ﾃﾞｰﾀ_OFF
OUT 711.07  ; R_RV_Low_(RT2)保持
; rung 27
LDNOT H10.04  ; ﾀﾞﾐｰ運転
AND 212.00  ; OV/RV_2CH_有り
LD H10.04  ; ﾀﾞﾐｰ運転
AND H10.10  ; RT_選択
ORLD
AND 520.08  ; R_RV_Hi(8)
@AND 700.01  ; 2CH_ﾃﾞｰﾀ取込
OR 711.08  ; R_RV_Hi_(RT2)保持
@ANDNOT 701.01  ; ﾃﾞｰﾀ_OFF
OUT 711.08  ; R_RV_Hi_(RT2)保持
; rung 28
LDNOT H10.04  ; ﾀﾞﾐｰ運転
AND 212.00  ; OV/RV_2CH_有り
LD H10.04  ; ﾀﾞﾐｰ運転
AND H10.10  ; RT_選択
ORLD
AND 520.10  ; ｺｲﾙ抵抗不良
@AND 700.01  ; 2CH_ﾃﾞｰﾀ取込
OR 711.10  ; 2CH_ｺｲﾙ抵抗不良
@ANDNOT 701.01  ; ﾃﾞｰﾀ_OFF
OUT 711.10  ; 2CH_ｺｲﾙ抵抗不良
; rung 29
LDNOT H10.04  ; ﾀﾞﾐｰ運転
AND 212.00  ; OV/RV_2CH_有り
LD H10.04  ; ﾀﾞﾐｰ運転
AND H10.10  ; RT_選択
ORLD
AND 520.11  ; ｺｲﾙ抵抗異常
@AND 700.01  ; 2CH_ﾃﾞｰﾀ取込
OR 711.11  ; 2CH_ｺｲﾙ抵抗NG
@ANDNOT 701.01  ; ﾃﾞｰﾀ_OFF
OUT 711.11  ; 2CH_ｺｲﾙ抵抗NG

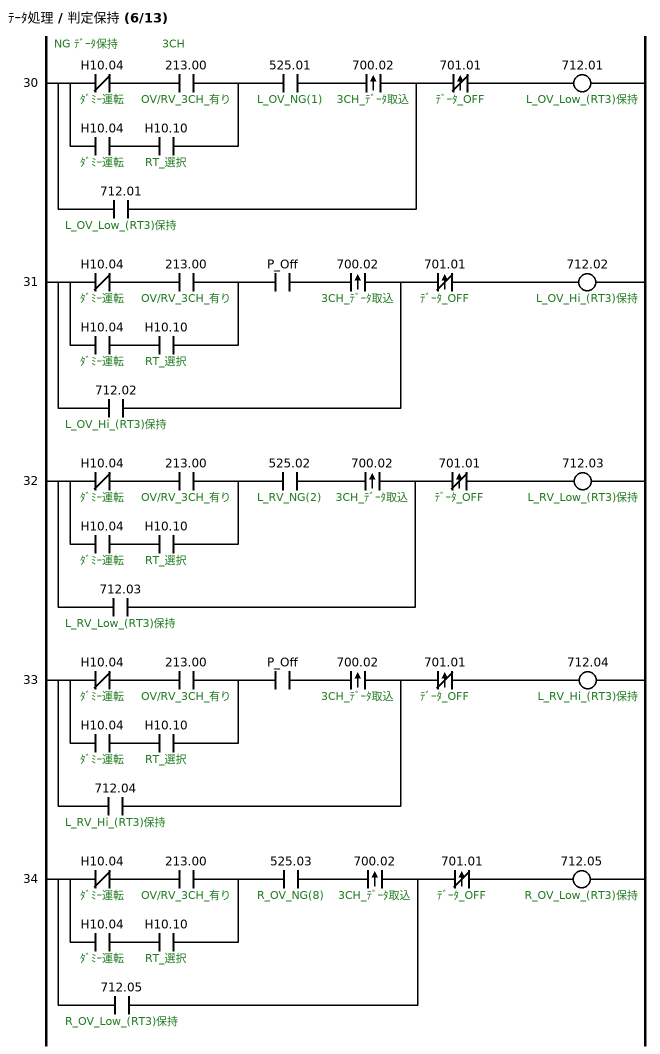
; rung 30: NG ﾃﾞｰﾀ保持　　　　3CH
LDNOT H10.04  ; ﾀﾞﾐｰ運転
AND 213.00  ; OV/RV_3CH_有り
LD H10.04  ; ﾀﾞﾐｰ運転
AND H10.10  ; RT_選択
ORLD
AND 525.01  ; L_OV_NG(1)
@AND 700.02  ; 3CH_ﾃﾞｰﾀ取込
OR 712.01  ; L_OV_Low_(RT3)保持
@ANDNOT 701.01  ; ﾃﾞｰﾀ_OFF
OUT 712.01  ; L_OV_Low_(RT3)保持
; rung 31
LDNOT H10.04  ; ﾀﾞﾐｰ運転
AND 213.00  ; OV/RV_3CH_有り
LD H10.04  ; ﾀﾞﾐｰ運転
AND H10.10  ; RT_選択
ORLD
AND P_Off
@AND 700.02  ; 3CH_ﾃﾞｰﾀ取込
OR 712.02  ; L_OV_Hi_(RT3)保持
@ANDNOT 701.01  ; ﾃﾞｰﾀ_OFF
OUT 712.02  ; L_OV_Hi_(RT3)保持
; rung 32
LDNOT H10.04  ; ﾀﾞﾐｰ運転
AND 213.00  ; OV/RV_3CH_有り
LD H10.04  ; ﾀﾞﾐｰ運転
AND H10.10  ; RT_選択
ORLD
AND 525.02  ; L_RV_NG(2)
@AND 700.02  ; 3CH_ﾃﾞｰﾀ取込
OR 712.03  ; L_RV_Low_(RT3)保持
@ANDNOT 701.01  ; ﾃﾞｰﾀ_OFF
OUT 712.03  ; L_RV_Low_(RT3)保持
; rung 33
LDNOT H10.04  ; ﾀﾞﾐｰ運転
AND 213.00  ; OV/RV_3CH_有り
LD H10.04  ; ﾀﾞﾐｰ運転
AND H10.10  ; RT_選択
ORLD
AND P_Off
@AND 700.02  ; 3CH_ﾃﾞｰﾀ取込
OR 712.04  ; L_RV_Hi_(RT3)保持
@ANDNOT 701.01  ; ﾃﾞｰﾀ_OFF
OUT 712.04  ; L_RV_Hi_(RT3)保持
; rung 34
LDNOT H10.04  ; ﾀﾞﾐｰ運転
AND 213.00  ; OV/RV_3CH_有り
LD H10.04  ; ﾀﾞﾐｰ運転
AND H10.10  ; RT_選択
ORLD
AND 525.03  ; R_OV_NG(8)
@AND 700.02  ; 3CH_ﾃﾞｰﾀ取込
OR 712.05  ; R_OV_Low_(RT3)保持
@ANDNOT 701.01  ; ﾃﾞｰﾀ_OFF
OUT 712.05  ; R_OV_Low_(RT3)保持

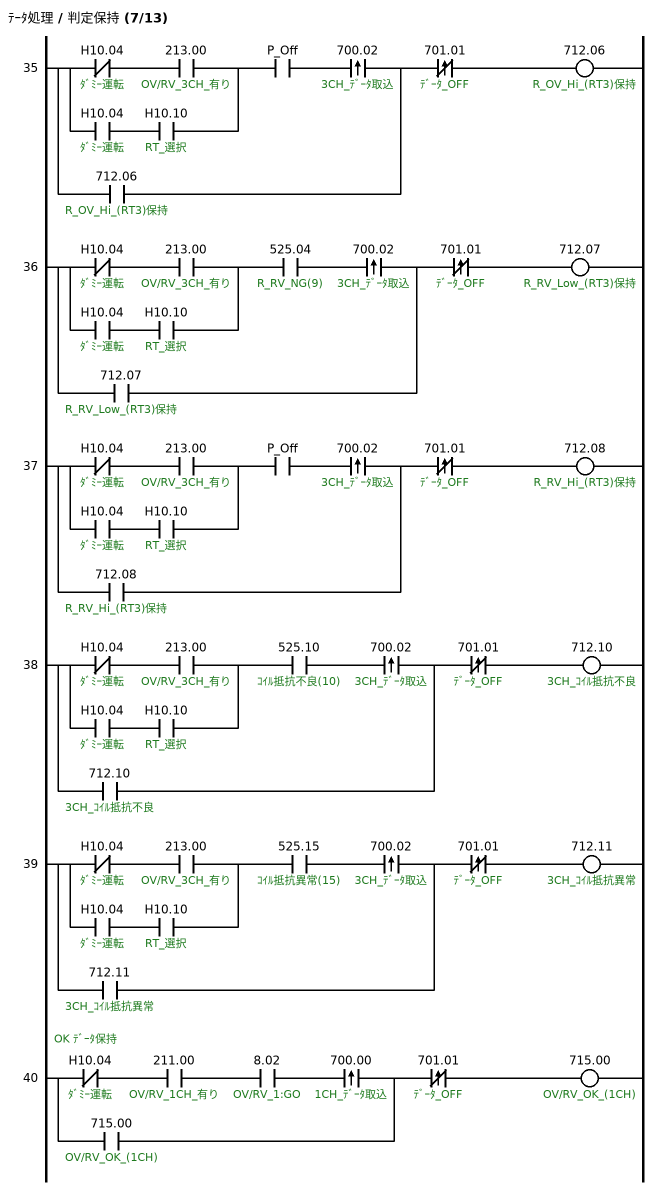
; rung 35
LDNOT H10.04  ; ﾀﾞﾐｰ運転
AND 213.00  ; OV/RV_3CH_有り
LD H10.04  ; ﾀﾞﾐｰ運転
AND H10.10  ; RT_選択
ORLD
AND P_Off
@AND 700.02  ; 3CH_ﾃﾞｰﾀ取込
OR 712.06  ; R_OV_Hi_(RT3)保持
@ANDNOT 701.01  ; ﾃﾞｰﾀ_OFF
OUT 712.06  ; R_OV_Hi_(RT3)保持
; rung 36
LDNOT H10.04  ; ﾀﾞﾐｰ運転
AND 213.00  ; OV/RV_3CH_有り
LD H10.04  ; ﾀﾞﾐｰ運転
AND H10.10  ; RT_選択
ORLD
AND 525.04  ; R_RV_NG(9)
@AND 700.02  ; 3CH_ﾃﾞｰﾀ取込
OR 712.07  ; R_RV_Low_(RT3)保持
@ANDNOT 701.01  ; ﾃﾞｰﾀ_OFF
OUT 712.07  ; R_RV_Low_(RT3)保持
; rung 37
LDNOT H10.04  ; ﾀﾞﾐｰ運転
AND 213.00  ; OV/RV_3CH_有り
LD H10.04  ; ﾀﾞﾐｰ運転
AND H10.10  ; RT_選択
ORLD
AND P_Off
@AND 700.02  ; 3CH_ﾃﾞｰﾀ取込
OR 712.08  ; R_RV_Hi_(RT3)保持
@ANDNOT 701.01  ; ﾃﾞｰﾀ_OFF
OUT 712.08  ; R_RV_Hi_(RT3)保持
; rung 38
LDNOT H10.04  ; ﾀﾞﾐｰ運転
AND 213.00  ; OV/RV_3CH_有り
LD H10.04  ; ﾀﾞﾐｰ運転
AND H10.10  ; RT_選択
ORLD
AND 525.10  ; ｺｲﾙ抵抗不良(10)
@AND 700.02  ; 3CH_ﾃﾞｰﾀ取込
OR 712.10  ; 3CH_ｺｲﾙ抵抗不良
@ANDNOT 701.01  ; ﾃﾞｰﾀ_OFF
OUT 712.10  ; 3CH_ｺｲﾙ抵抗不良
; rung 39
LDNOT H10.04  ; ﾀﾞﾐｰ運転
AND 213.00  ; OV/RV_3CH_有り
LD H10.04  ; ﾀﾞﾐｰ運転
AND H10.10  ; RT_選択
ORLD
AND 525.15  ; ｺｲﾙ抵抗異常(15)
@AND 700.02  ; 3CH_ﾃﾞｰﾀ取込
OR 712.11  ; 3CH_ｺｲﾙ抵抗異常
@ANDNOT 701.01  ; ﾃﾞｰﾀ_OFF
OUT 712.11  ; 3CH_ｺｲﾙ抵抗異常
; rung 40: OK ﾃﾞｰﾀ保持
LDNOT H10.04  ; ﾀﾞﾐｰ運転
AND 211.00  ; OV/RV_1CH_有り
AND 8.02  ; OV/RV_1:GO
@AND 700.00  ; 1CH_ﾃﾞｰﾀ取込
OR 715.00  ; OV/RV_OK_(1CH)
@ANDNOT 701.01  ; ﾃﾞｰﾀ_OFF
OUT 715.00  ; OV/RV_OK_(1CH)

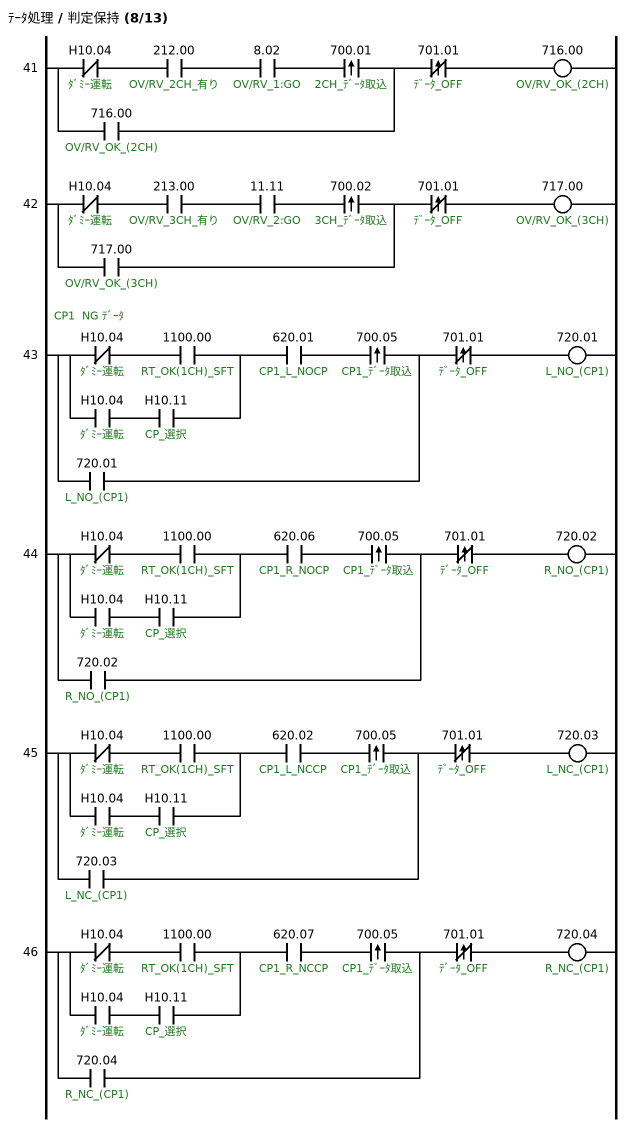
; rung 41
LDNOT H10.04  ; ﾀﾞﾐｰ運転
AND 212.00  ; OV/RV_2CH_有り
AND 8.02  ; OV/RV_1:GO
@AND 700.01  ; 2CH_ﾃﾞｰﾀ取込
OR 716.00  ; OV/RV_OK_(2CH)
@ANDNOT 701.01  ; ﾃﾞｰﾀ_OFF
OUT 716.00  ; OV/RV_OK_(2CH)
; rung 42
LDNOT H10.04  ; ﾀﾞﾐｰ運転
AND 213.00  ; OV/RV_3CH_有り
AND 11.11  ; OV/RV_2:GO
@AND 700.02  ; 3CH_ﾃﾞｰﾀ取込
OR 717.00  ; OV/RV_OK_(3CH)
@ANDNOT 701.01  ; ﾃﾞｰﾀ_OFF
OUT 717.00  ; OV/RV_OK_(3CH)
; rung 43: CP1  NG ﾃﾞｰﾀ
LDNOT H10.04  ; ﾀﾞﾐｰ運転
AND 1100.00  ; RT_OK(1CH)_SFT
LD H10.04  ; ﾀﾞﾐｰ運転
AND H10.11  ; CP_選択
ORLD
AND 620.01  ; CP1_L_NOCP
@AND 700.05  ; CP1_ﾃﾞｰﾀ取込
OR 720.01  ; L_NO_(CP1)
@ANDNOT 701.01  ; ﾃﾞｰﾀ_OFF
OUT 720.01  ; L_NO_(CP1)
; rung 44
LDNOT H10.04  ; ﾀﾞﾐｰ運転
AND 1100.00  ; RT_OK(1CH)_SFT
LD H10.04  ; ﾀﾞﾐｰ運転
AND H10.11  ; CP_選択
ORLD
AND 620.06  ; CP1_R_NOCP
@AND 700.05  ; CP1_ﾃﾞｰﾀ取込
OR 720.02  ; R_NO_(CP1)
@ANDNOT 701.01  ; ﾃﾞｰﾀ_OFF
OUT 720.02  ; R_NO_(CP1)
; rung 45
LDNOT H10.04  ; ﾀﾞﾐｰ運転
AND 1100.00  ; RT_OK(1CH)_SFT
LD H10.04  ; ﾀﾞﾐｰ運転
AND H10.11  ; CP_選択
ORLD
AND 620.02  ; CP1_L_NCCP
@AND 700.05  ; CP1_ﾃﾞｰﾀ取込
OR 720.03  ; L_NC_(CP1)
@ANDNOT 701.01  ; ﾃﾞｰﾀ_OFF
OUT 720.03  ; L_NC_(CP1)
; rung 46
LDNOT H10.04  ; ﾀﾞﾐｰ運転
AND 1100.00  ; RT_OK(1CH)_SFT
LD H10.04  ; ﾀﾞﾐｰ運転
AND H10.11  ; CP_選択
ORLD
AND 620.07  ; CP1_R_NCCP
@AND 700.05  ; CP1_ﾃﾞｰﾀ取込
OR 720.04  ; R_NC_(CP1)
@ANDNOT 701.01  ; ﾃﾞｰﾀ_OFF
OUT 720.04  ; R_NC_(CP1)

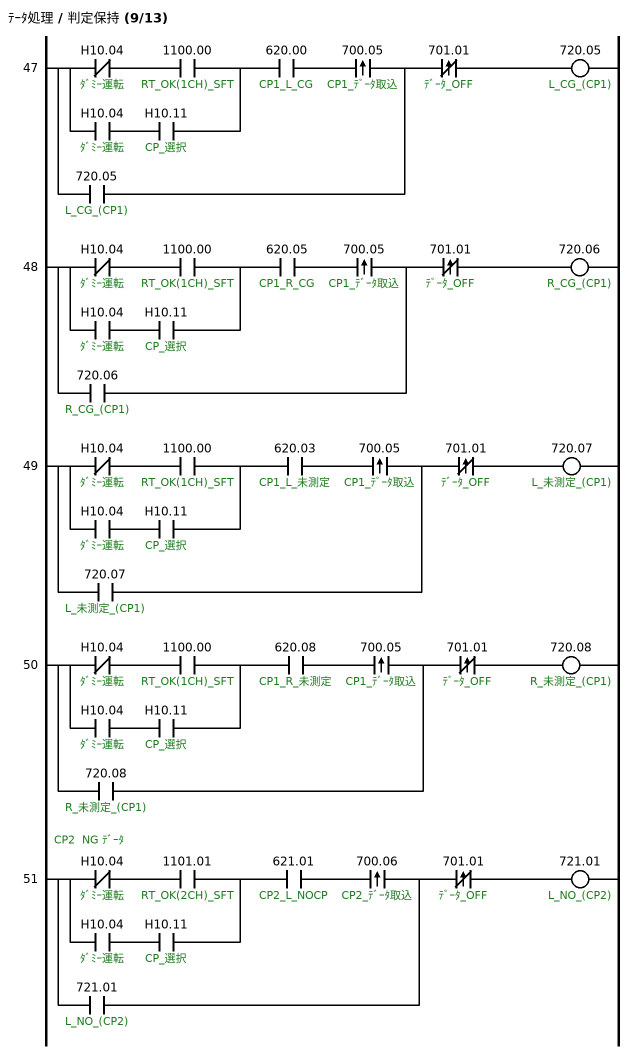
; rung 47
LDNOT H10.04  ; ﾀﾞﾐｰ運転
AND 1100.00  ; RT_OK(1CH)_SFT
LD H10.04  ; ﾀﾞﾐｰ運転
AND H10.11  ; CP_選択
ORLD
AND 620.00  ; CP1_L_CG
@AND 700.05  ; CP1_ﾃﾞｰﾀ取込
OR 720.05  ; L_CG_(CP1)
@ANDNOT 701.01  ; ﾃﾞｰﾀ_OFF
OUT 720.05  ; L_CG_(CP1)
; rung 48
LDNOT H10.04  ; ﾀﾞﾐｰ運転
AND 1100.00  ; RT_OK(1CH)_SFT
LD H10.04  ; ﾀﾞﾐｰ運転
AND H10.11  ; CP_選択
ORLD
AND 620.05  ; CP1_R_CG
@AND 700.05  ; CP1_ﾃﾞｰﾀ取込
OR 720.06  ; R_CG_(CP1)
@ANDNOT 701.01  ; ﾃﾞｰﾀ_OFF
OUT 720.06  ; R_CG_(CP1)
; rung 49
LDNOT H10.04  ; ﾀﾞﾐｰ運転
AND 1100.00  ; RT_OK(1CH)_SFT
LD H10.04  ; ﾀﾞﾐｰ運転
AND H10.11  ; CP_選択
ORLD
AND 620.03  ; CP1_L_未測定
@AND 700.05  ; CP1_ﾃﾞｰﾀ取込
OR 720.07  ; L_未測定_(CP1)
@ANDNOT 701.01  ; ﾃﾞｰﾀ_OFF
OUT 720.07  ; L_未測定_(CP1)
; rung 50
LDNOT H10.04  ; ﾀﾞﾐｰ運転
AND 1100.00  ; RT_OK(1CH)_SFT
LD H10.04  ; ﾀﾞﾐｰ運転
AND H10.11  ; CP_選択
ORLD
AND 620.08  ; CP1_R_未測定
@AND 700.05  ; CP1_ﾃﾞｰﾀ取込
OR 720.08  ; R_未測定_(CP1)
@ANDNOT 701.01  ; ﾃﾞｰﾀ_OFF
OUT 720.08  ; R_未測定_(CP1)
; rung 51: CP2  NG ﾃﾞｰﾀ
LDNOT H10.04  ; ﾀﾞﾐｰ運転
AND 1101.01  ; RT_OK(2CH)_SFT
LD H10.04  ; ﾀﾞﾐｰ運転
AND H10.11  ; CP_選択
ORLD
AND 621.01  ; CP2_L_NOCP
@AND 700.06  ; CP2_ﾃﾞｰﾀ取込
OR 721.01  ; L_NO_(CP2)
@ANDNOT 701.01  ; ﾃﾞｰﾀ_OFF
OUT 721.01  ; L_NO_(CP2)

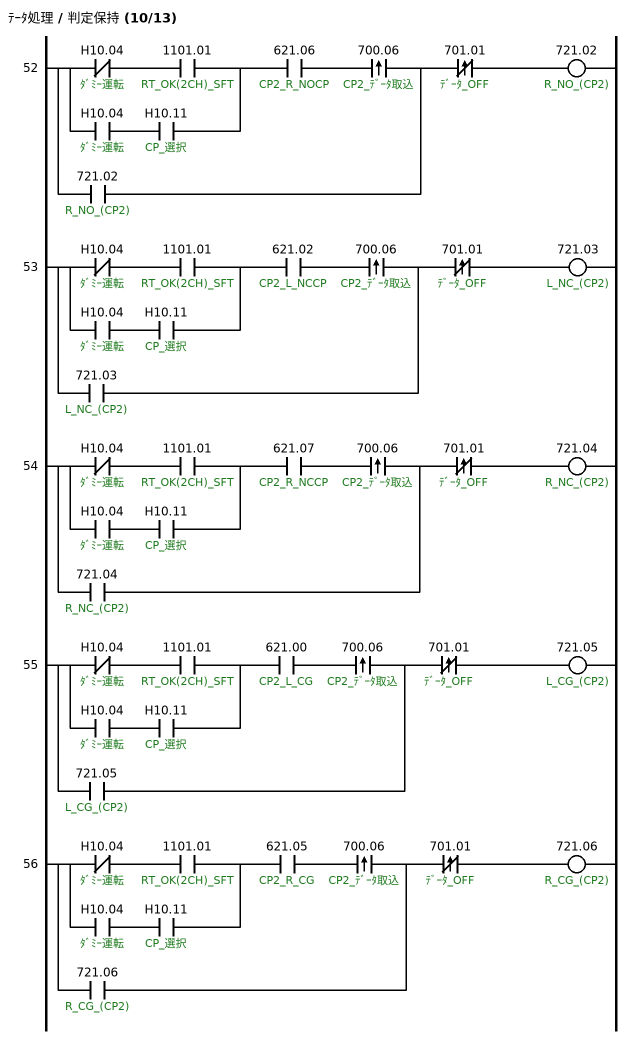
; rung 52
LDNOT H10.04  ; ﾀﾞﾐｰ運転
AND 1101.01  ; RT_OK(2CH)_SFT
LD H10.04  ; ﾀﾞﾐｰ運転
AND H10.11  ; CP_選択
ORLD
AND 621.06  ; CP2_R_NOCP
@AND 700.06  ; CP2_ﾃﾞｰﾀ取込
OR 721.02  ; R_NO_(CP2)
@ANDNOT 701.01  ; ﾃﾞｰﾀ_OFF
OUT 721.02  ; R_NO_(CP2)
; rung 53
LDNOT H10.04  ; ﾀﾞﾐｰ運転
AND 1101.01  ; RT_OK(2CH)_SFT
LD H10.04  ; ﾀﾞﾐｰ運転
AND H10.11  ; CP_選択
ORLD
AND 621.02  ; CP2_L_NCCP
@AND 700.06  ; CP2_ﾃﾞｰﾀ取込
OR 721.03  ; L_NC_(CP2)
@ANDNOT 701.01  ; ﾃﾞｰﾀ_OFF
OUT 721.03  ; L_NC_(CP2)
; rung 54
LDNOT H10.04  ; ﾀﾞﾐｰ運転
AND 1101.01  ; RT_OK(2CH)_SFT
LD H10.04  ; ﾀﾞﾐｰ運転
AND H10.11  ; CP_選択
ORLD
AND 621.07  ; CP2_R_NCCP
@AND 700.06  ; CP2_ﾃﾞｰﾀ取込
OR 721.04  ; R_NC_(CP2)
@ANDNOT 701.01  ; ﾃﾞｰﾀ_OFF
OUT 721.04  ; R_NC_(CP2)
; rung 55
LDNOT H10.04  ; ﾀﾞﾐｰ運転
AND 1101.01  ; RT_OK(2CH)_SFT
LD H10.04  ; ﾀﾞﾐｰ運転
AND H10.11  ; CP_選択
ORLD
AND 621.00  ; CP2_L_CG
@AND 700.06  ; CP2_ﾃﾞｰﾀ取込
OR 721.05  ; L_CG_(CP2)
@ANDNOT 701.01  ; ﾃﾞｰﾀ_OFF
OUT 721.05  ; L_CG_(CP2)
; rung 56
LDNOT H10.04  ; ﾀﾞﾐｰ運転
AND 1101.01  ; RT_OK(2CH)_SFT
LD H10.04  ; ﾀﾞﾐｰ運転
AND H10.11  ; CP_選択
ORLD
AND 621.05  ; CP2_R_CG
@AND 700.06  ; CP2_ﾃﾞｰﾀ取込
OR 721.06  ; R_CG_(CP2)
@ANDNOT 701.01  ; ﾃﾞｰﾀ_OFF
OUT 721.06  ; R_CG_(CP2)

